(* IEC 61131-3 sources: Industry-PLC-LLM/data/PLCBEAD_repo/PLCBEAD_PLCEmbed-main/PLC-BEAD/Source/GEB/LINEAR_INT, 1 file *)

(* ---- LINEAR_INT.ST ---- *)
TYPE
	oscat_ARRAY_X               : ARRAY [0..1]    OF REAL;
	oscat_XY                    : ARRAY [1..20]   OF oscat_ARRAY_X;
END_TYPE

FUNCTION_BLOCK LINEAR_INT_Block

	VAR_INPUT
		X :	REAL;
		XY :	oscat_XY;
		PTS :	INT;
	END_VAR

	VAR_OUTPUT
		LINEAR_INT :	REAL;
	END_VAR

	VAR
		i :	INT;
		i2 :	INT;
		PTSS :	INT;
	END_VAR

	PTSS := PTS;
	PTSS := MIN(PTSS,20);

	i := 2;

	WHILE (i < PTS) AND (XY[i][0] < X) DO
		i := i + 1;
	END_WHILE;

	i2 := i-1;

	LINEAR_INT := ((XY[i][1] - XY[i2][1]) * X - XY[i][1] * XY[i2][0] + XY[i2][1] * XY[i][0]) / (XY[i][0] - XY[i2][0]);

END_FUNCTION_BLOCK

PROGRAM program0

	VAR
		X :	REAL;
		XY :	oscat_XY;
		PTS :	INT;

		LINEAR_INT :	REAL;

		func_block : LINEAR_INT_Block;
	END_VAR
	func_block.X := X;
	func_block.XY := XY;
	func_block.PTS := PTS;

	func_block();
	LINEAR_INT := func_block.LINEAR_INT;

END_PROGRAM
